// TIA Portal project "Lab4" (V16)

(* hardware
DEVICE "S71500/ET200MP station_1"  S7-1500 station
   slot 0: "PM 190W 120/230VAC"  PM 190W 120/230VAC  6EP1333-4BA00
   slot 0: "Perfil soporte_0"  Rack  6ES7 590-1***0-0AA0
   slot 1: "PLC_1"  CPU 1516-3 PN/DP  6ES7 516-3AN01-0AB0  V1.8
      slot 3: "Display de la CPU_1"  6ES7591-1BA00-0AA0
      slot 32768: "Interfaz PROFINET_1"  X1
         slot 32769: "Puerto_1"  X1 P1
         slot 32770: "Puerto_2"  X1 P2
      slot 33024: "Interfaz PROFINET_2"  X2
         slot 33025: "Puerto_1"  X2 P1
      slot 33280: "Interfaz DP_1"  X3
   slot 2: "DI 32x24VDC HF_1"  DI 32x24VDC HF  6ES7 521-1BL00-0AB0  V1.0
   slot 3: "DQ 32x24VDC/0.5A ST_1"  DQ 32x24VDC/0.5A ST  6ES7 522-1BL00-0AB0  V1.0
   slot 4: "AI 8xU/I/RTD/TC ST_1"  AI 8xU/I/RTD/TC ST  6ES7 531-7KF00-0AB0  V1.0
   slot 5: "AQ 4xU/I ST_1"  AQ 4xU/I ST  6ES7 532-5HD00-0AB0  V1.0
*)

// ===== PLC "PLC_1"  CPU 1516-3 PN/DP =====

VAR_GLOBAL   // PLC tag table "Tabla de variables estándar"
   "10001" AT %M0.0 : Bool;
   "10003" AT %M0.2 : Bool;
   "ON2" AT %M100.0 : Bool;
   "10005" AT %M0.4 : Bool;
   "OFF14-15-ONMP1-CUA" AT %M201.0 : Bool;
   "OFFMP1-CUA" AT %M202.0 : Bool;
   "OFFMP2YONMP1-C1" AT %M212.0 : Bool;
   "ON1YON4" AT %M101.0 : Bool;
   "10004" AT %M0.3 : Bool;
   "OFF1YOFF4" AT %M102.0 : Bool;
   "OFF2" AT %M103.0 : Bool;
   "ON1YON3" AT %M104.0 : Bool;
   "OFF1YON4" AT %M105.0 : Bool;
   "OFF3YOFF4" AT %M106.0 : Bool;
   "2" AT %Q0.1 : Bool;
   "1" AT %Q0.0 : Bool;
   "4" AT %Q0.3 : Bool;
   "3" AT %Q0.2 : Bool;
   "10002" AT %M0.1 : Bool;
   "10006" AT %M0.5 : Bool;
   "10028" AT %I0.0 : Bool;
   "10021" AT %I0.4 : Bool;
   "10023" AT %I0.1 : Bool;
   "10025" AT %I0.5 : Bool;
   "ON9-10-15" AT %M210.0 : Bool;
   "OFF8" AT %M116.0 : Bool;
   "OFFMP1-C1" AT %M213.0 : Bool;
   "10" AT %Q1.0 : Bool;
   "9" AT %Q0.7 : Bool;
   "15" AT %Q1.5 : Bool;
   "10010" AT %M0.7 : Bool;
   "10011" AT %M1.0 : Bool;
   "10012" AT %M1.1 : Bool;
   "10009" AT %M0.6 : Bool;
   "OFF9-10-15YONMP2-C1" AT %M211.0 : Bool;
   "OFF15-13-12-11YONMP2-C2" AT %M216.0 : Bool;
   "ON8YON5" AT %M110.0 : Bool;
   "OFF8YOFF5" AT %M111.0 : Bool;
   "ON6" AT %M112.0 : Bool;
   "ON5" AT %M113.0 : Bool;
   "ON8YOFF5" AT %M114.0 : Bool;
   "OFF6" AT %M115.0 : Bool;
   "5" AT %Q0.4 : Bool;
   "8" AT %Q0.6 : Bool;
   "6" AT %Q0.5 : Bool;
   "10022" AT %I0.3 : Bool;
   "14" AT %Q1.4 : Bool;
   "ON14-15" AT %M200.0 : Bool;
   "10024" AT %I0.2 : Bool;
   "ON15-11-12-13" AT %M215.0 : Bool;
   "OFFMP1-C2" AT %M218.0 : Bool;
   "OFFMP2YONMP1-C2" AT %M217.0 : Bool;
   "11" AT %Q1.1 : Bool;
   "12" AT %Q1.2 : Bool;
   "13" AT %Q1.3 : Bool;
   "RUN" AT %M2.0 : Bool;
   "STOP" AT %M2.1 : Bool;
   "Inic_Proce" AT %M60.0 : Bool;
   "Sec_Cuadrado" AT %M60.1 : Bool;
   "Aux1" AT %M300.0 : Bool;
   "Sec_Cilindro1" AT %M60.2 : Bool;
   "Sec_Cilindro2" AT %M60.3 : Bool;
   "Aux2" AT %M300.1 : Bool;
   "15AUX" AT %M500.0 : Bool;
   "Tag_1" AT %MB3 : Byte;
END_VAR

// folder: System blocks/Program resources

DATA_BLOCK "IEC_Counter_0_DB"   // DB1
{ S7_Optimized_Access := 'TRUE' }
AUTHOR : Simatic
FAMILY : IEC
NAME : CNTR
VERSION : 1.0
// stored: InstanceOfName IEC_COUNTER
"IEC_COUNTER"
BEGIN
END_DATA_BLOCK

// folder: (top level)

FUNCTION "MP1" : Void   // FC1, LAD
{ S7_Optimized_Access := 'TRUE' }
VERSION : 0.1
BEGIN

REGION Network 1
   // MP1
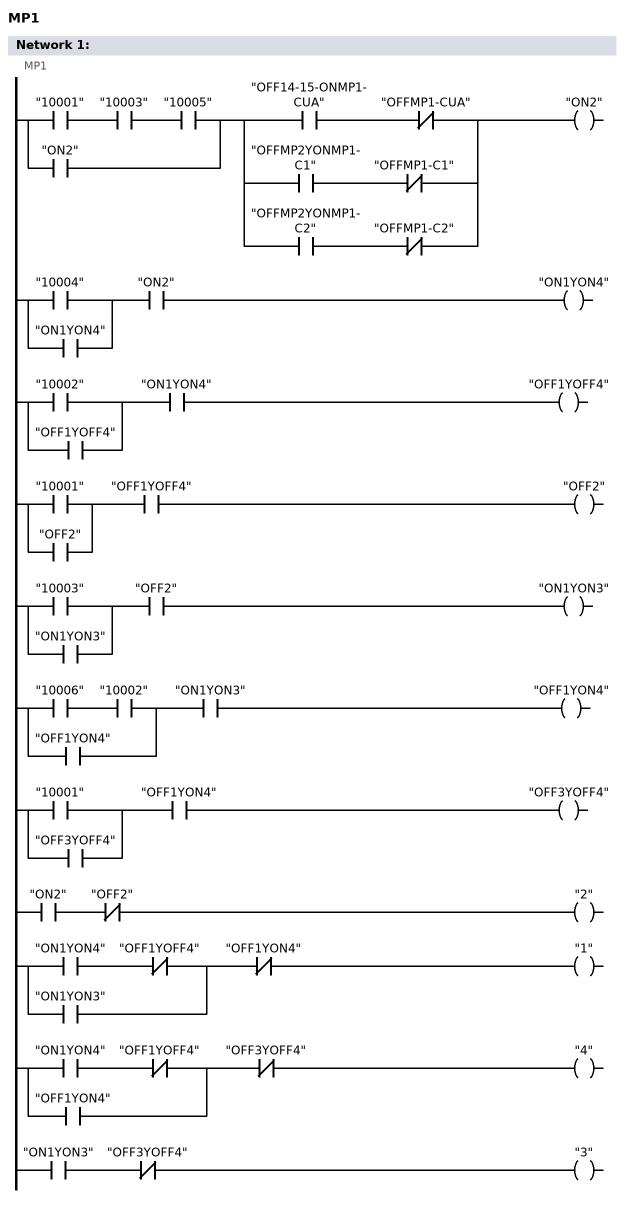
   RUNG wire#powerrail
      Contact( "10001" )
      Contact( "10003" )
      Contact( "10005" )
      wire#w1
      Contact( "OFF14-15-ONMP1-CUA" )
      I_Contact( "OFFMP1-CUA" )
      wire#w2
      Coil( "ON2" )
   END_RUNG
   RUNG wire#powerrail
      Contact( "ON2" )
   END_RUNG wire#w1
   RUNG wire#w1
      Contact( "OFFMP2YONMP1-C1" )
      I_Contact( "OFFMP1-C1" )
   END_RUNG wire#w2
   RUNG wire#w1
      Contact( "OFFMP2YONMP1-C2" )
      I_Contact( "OFFMP1-C2" )
   END_RUNG wire#w2
   RUNG wire#powerrail
      Contact( "10004" )
      wire#w3
      Contact( "ON2" )
      Coil( "ON1YON4" )
   END_RUNG
   RUNG wire#powerrail
      Contact( "ON1YON4" )
   END_RUNG wire#w3
   RUNG wire#powerrail
      Contact( "10002" )
      wire#w4
      Contact( "ON1YON4" )
      Coil( "OFF1YOFF4" )
   END_RUNG
   RUNG wire#powerrail
      Contact( "OFF1YOFF4" )
   END_RUNG wire#w4
   RUNG wire#powerrail
      Contact( "10001" )
      wire#w5
      Contact( "OFF1YOFF4" )
      Coil( "OFF2" )
   END_RUNG
   RUNG wire#powerrail
      Contact( "OFF2" )
   END_RUNG wire#w5
   RUNG wire#powerrail
      Contact( "10003" )
      wire#w6
      Contact( "OFF2" )
      Coil( "ON1YON3" )
   END_RUNG
   RUNG wire#powerrail
      Contact( "ON1YON3" )
   END_RUNG wire#w6
   RUNG wire#powerrail
      Contact( "10006" )
      Contact( "10002" )
      wire#w7
      Contact( "ON1YON3" )
      Coil( "OFF1YON4" )
   END_RUNG
   RUNG wire#powerrail
      Contact( "OFF1YON4" )
   END_RUNG wire#w7
   RUNG wire#powerrail
      Contact( "10001" )
      wire#w8
      Contact( "OFF1YON4" )
      Coil( "OFF3YOFF4" )
   END_RUNG
   RUNG wire#powerrail
      Contact( "OFF3YOFF4" )
   END_RUNG wire#w8
   RUNG wire#powerrail
      Contact( "ON2" )
      I_Contact( "OFF2" )
      Coil( "2" )
   END_RUNG
   RUNG wire#powerrail
      Contact( "ON1YON4" )
      I_Contact( "OFF1YOFF4" )
      wire#w9
      I_Contact( "OFF1YON4" )
      Coil( "1" )
   END_RUNG
   RUNG wire#powerrail
      Contact( "ON1YON3" )
   END_RUNG wire#w9
   RUNG wire#powerrail
      Contact( "ON1YON4" )
      I_Contact( "OFF1YOFF4" )
      wire#w10
      I_Contact( "OFF3YOFF4" )
      Coil( "4" )
   END_RUNG
   RUNG wire#powerrail
      Contact( "OFF1YON4" )
   END_RUNG wire#w10
   RUNG wire#powerrail
      Contact( "ON1YON3" )
      I_Contact( "OFF3YOFF4" )
      Coil( "3" )
   END_RUNG
   // the same network as SCL:
   "ON2" := (("10001" AND "10003" AND "10005") OR "ON2") AND (("OFF14-15-ONMP1-CUA" AND NOT "OFFMP1-CUA") OR ("OFFMP2YONMP1-C1" AND NOT "OFFMP1-C1") OR ("OFFMP2YONMP1-C2" AND NOT "OFFMP1-C2"));
   "ON1YON4" := ("10004" OR "ON1YON4") AND "ON2";
   "OFF1YOFF4" := ("10002" OR "OFF1YOFF4") AND "ON1YON4";
   "OFF2" := ("10001" OR "OFF2") AND "OFF1YOFF4";
   "ON1YON3" := ("10003" OR "ON1YON3") AND "OFF2";
   "OFF1YON4" := (("10006" AND "10002") OR "OFF1YON4") AND "ON1YON3";
   "OFF3YOFF4" := ("10001" OR "OFF3YOFF4") AND "OFF1YON4";
   "2" := "ON2" AND NOT "OFF2";
   "1" := (("ON1YON4" AND NOT "OFF1YOFF4") OR "ON1YON3") AND NOT "OFF1YON4";
   "4" := (("ON1YON4" AND NOT "OFF1YOFF4") OR "OFF1YON4") AND NOT "OFF3YOFF4";
   "3" := "ON1YON3" AND NOT "OFF3YOFF4";
END_REGION
END_FUNCTION

FUNCTION "MP2" : Void   // FC2, LAD
{ S7_Optimized_Access := 'TRUE' }
VERSION : 0.1
BEGIN

REGION Network 1
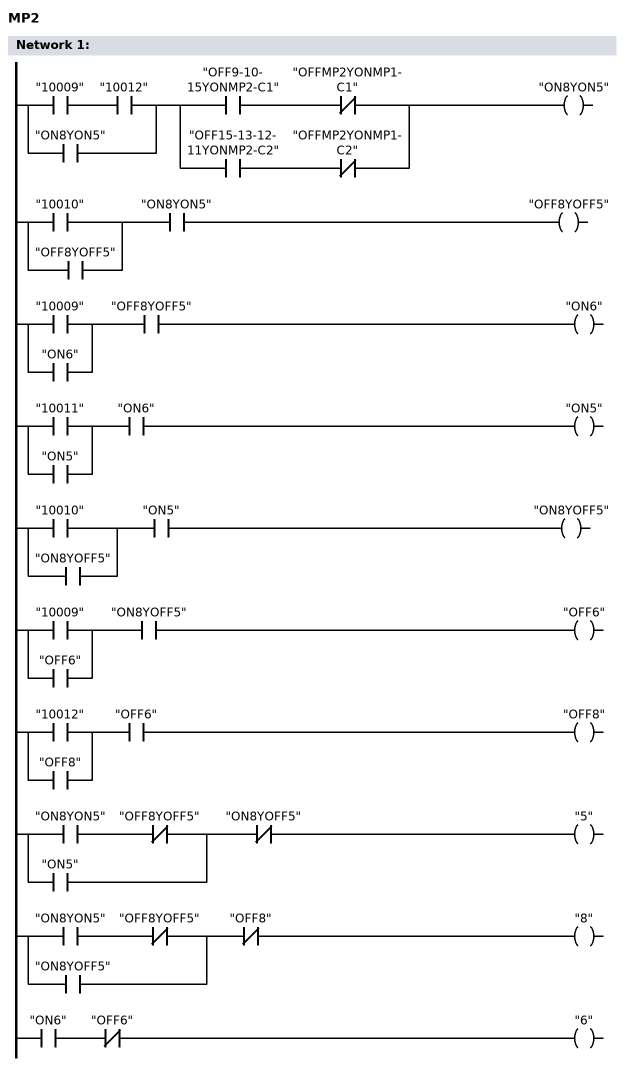
   RUNG wire#powerrail
      Contact( "10009" )
      Contact( "10012" )
      wire#w1
      Contact( "OFF9-10-15YONMP2-C1" )
      I_Contact( "OFFMP2YONMP1-C1" )
      wire#w2
      Coil( "ON8YON5" )
   END_RUNG
   RUNG wire#powerrail
      Contact( "ON8YON5" )
   END_RUNG wire#w1
   RUNG wire#w1
      Contact( "OFF15-13-12-11YONMP2-C2" )
      I_Contact( "OFFMP2YONMP1-C2" )
   END_RUNG wire#w2
   RUNG wire#powerrail
      Contact( "10010" )
      wire#w3
      Contact( "ON8YON5" )
      Coil( "OFF8YOFF5" )
   END_RUNG
   RUNG wire#powerrail
      Contact( "OFF8YOFF5" )
   END_RUNG wire#w3
   RUNG wire#powerrail
      Contact( "10009" )
      wire#w4
      Contact( "OFF8YOFF5" )
      Coil( "ON6" )
   END_RUNG
   RUNG wire#powerrail
      Contact( "ON6" )
   END_RUNG wire#w4
   RUNG wire#powerrail
      Contact( "10011" )
      wire#w5
      Contact( "ON6" )
      Coil( "ON5" )
   END_RUNG
   RUNG wire#powerrail
      Contact( "ON5" )
   END_RUNG wire#w5
   RUNG wire#powerrail
      Contact( "10010" )
      wire#w6
      Contact( "ON5" )
      Coil( "ON8YOFF5" )
   END_RUNG
   RUNG wire#powerrail
      Contact( "ON8YOFF5" )
   END_RUNG wire#w6
   RUNG wire#powerrail
      Contact( "10009" )
      wire#w7
      Contact( "ON8YOFF5" )
      Coil( "OFF6" )
   END_RUNG
   RUNG wire#powerrail
      Contact( "OFF6" )
   END_RUNG wire#w7
   RUNG wire#powerrail
      Contact( "10012" )
      wire#w8
      Contact( "OFF6" )
      Coil( "OFF8" )
   END_RUNG
   RUNG wire#powerrail
      Contact( "OFF8" )
   END_RUNG wire#w8
   RUNG wire#powerrail
      Contact( "ON8YON5" )
      I_Contact( "OFF8YOFF5" )
      wire#w9
      I_Contact( "ON8YOFF5" )
      Coil( "5" )
   END_RUNG
   RUNG wire#powerrail
      Contact( "ON5" )
   END_RUNG wire#w9
   RUNG wire#powerrail
      Contact( "ON8YON5" )
      I_Contact( "OFF8YOFF5" )
      wire#w10
      I_Contact( "OFF8" )
      Coil( "8" )
   END_RUNG
   RUNG wire#powerrail
      Contact( "ON8YOFF5" )
   END_RUNG wire#w10
   RUNG wire#powerrail
      Contact( "ON6" )
      I_Contact( "OFF6" )
      Coil( "6" )
   END_RUNG
   // the same network as SCL:
   "ON8YON5" := (("10009" AND "10012") OR "ON8YON5") AND (("OFF9-10-15YONMP2-C1" AND NOT "OFFMP2YONMP1-C1") OR ("OFF15-13-12-11YONMP2-C2" AND NOT "OFFMP2YONMP1-C2"));
   "OFF8YOFF5" := ("10010" OR "OFF8YOFF5") AND "ON8YON5";
   "ON6" := ("10009" OR "ON6") AND "OFF8YOFF5";
   "ON5" := ("10011" OR "ON5") AND "ON6";
   "ON8YOFF5" := ("10010" OR "ON8YOFF5") AND "ON5";
   "OFF6" := ("10009" OR "OFF6") AND "ON8YOFF5";
   "OFF8" := ("10012" OR "OFF8") AND "OFF6";
   "5" := (("ON8YON5" AND NOT "OFF8YOFF5") OR "ON5") AND NOT "ON8YOFF5";
   "8" := (("ON8YON5" AND NOT "OFF8YOFF5") OR "ON8YOFF5") AND NOT "OFF8";
   "6" := "ON6" AND NOT "OFF6";
END_REGION
END_FUNCTION

FUNCTION "CUADRADOS" : Void   // FC3, LAD
{ S7_Optimized_Access := 'TRUE' }
VERSION : 0.1
BEGIN

REGION Network 1
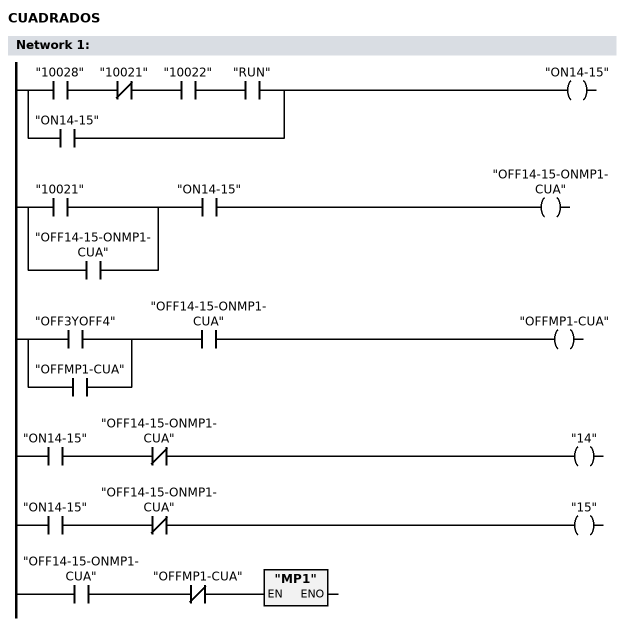
   RUNG wire#powerrail
      Contact( "10028" )
      I_Contact( "10021" )
      Contact( "10022" )
      Contact( "RUN" )
      wire#w1
      Coil( "ON14-15" )
   END_RUNG
   RUNG wire#powerrail
      Contact( "ON14-15" )
   END_RUNG wire#w1
   RUNG wire#powerrail
      Contact( "10021" )
      wire#w2
      Contact( "ON14-15" )
      Coil( "OFF14-15-ONMP1-CUA" )
   END_RUNG
   RUNG wire#powerrail
      Contact( "OFF14-15-ONMP1-CUA" )
   END_RUNG wire#w2
   RUNG wire#powerrail
      Contact( "OFF3YOFF4" )
      wire#w3
      Contact( "OFF14-15-ONMP1-CUA" )
      Coil( "OFFMP1-CUA" )
   END_RUNG
   RUNG wire#powerrail
      Contact( "OFFMP1-CUA" )
   END_RUNG wire#w3
   RUNG wire#powerrail
      Contact( "ON14-15" )
      I_Contact( "OFF14-15-ONMP1-CUA" )
      Coil( "14" )
   END_RUNG
   RUNG wire#powerrail
      Contact( "ON14-15" )
      I_Contact( "OFF14-15-ONMP1-CUA" )
      Coil( "15" )
   END_RUNG
   RUNG wire#powerrail
      Contact( "OFF14-15-ONMP1-CUA" )
      I_Contact( "OFFMP1-CUA" )
      "MP1"()
   END_RUNG
   // the same network as SCL:
   "ON14-15" := ("10028" AND NOT "10021" AND "10022" AND "RUN") OR "ON14-15";
   "OFF14-15-ONMP1-CUA" := ("10021" OR "OFF14-15-ONMP1-CUA") AND "ON14-15";
   "OFFMP1-CUA" := ("OFF3YOFF4" OR "OFFMP1-CUA") AND "OFF14-15-ONMP1-CUA";
   "14" := "ON14-15" AND NOT "OFF14-15-ONMP1-CUA";
   "15" := "ON14-15" AND NOT "OFF14-15-ONMP1-CUA";
   IF "OFF14-15-ONMP1-CUA" AND NOT "OFFMP1-CUA" THEN "MP1"(); END_IF;
END_REGION
END_FUNCTION

FUNCTION "CILINDRO1" : Void   // FC4, LAD
{ S7_Optimized_Access := 'TRUE' }
VERSION : 0.1
BEGIN

REGION Network 1
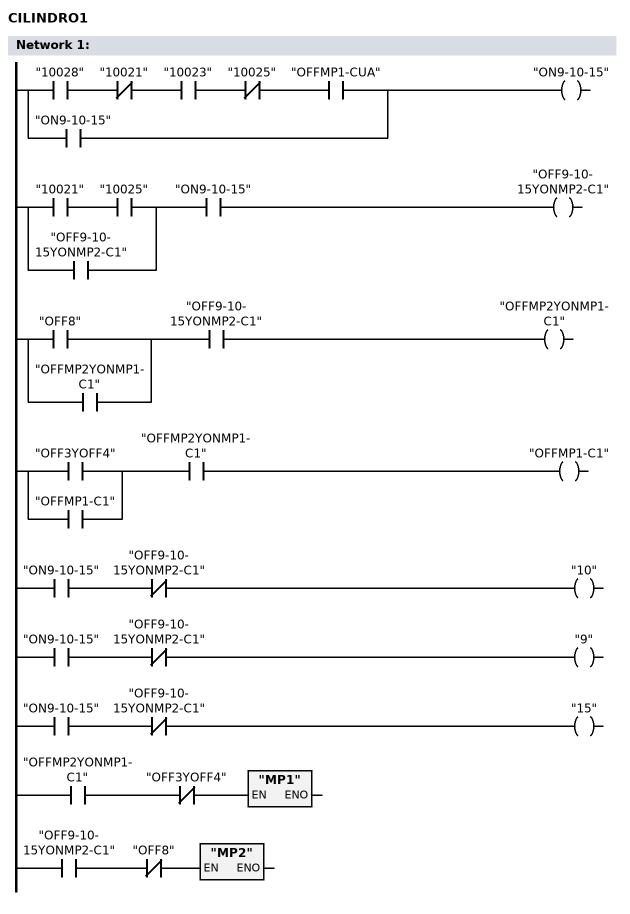
   RUNG wire#powerrail
      Contact( "10028" )
      I_Contact( "10021" )
      Contact( "10023" )
      I_Contact( "10025" )
      Contact( "OFFMP1-CUA" )
      wire#w1
      Coil( "ON9-10-15" )
   END_RUNG
   RUNG wire#powerrail
      Contact( "ON9-10-15" )
   END_RUNG wire#w1
   RUNG wire#powerrail
      Contact( "10021" )
      Contact( "10025" )
      wire#w2
      Contact( "ON9-10-15" )
      Coil( "OFF9-10-15YONMP2-C1" )
   END_RUNG
   RUNG wire#powerrail
      Contact( "OFF9-10-15YONMP2-C1" )
   END_RUNG wire#w2
   RUNG wire#powerrail
      Contact( "OFF8" )
      wire#w3
      Contact( "OFF9-10-15YONMP2-C1" )
      Coil( "OFFMP2YONMP1-C1" )
   END_RUNG
   RUNG wire#powerrail
      Contact( "OFFMP2YONMP1-C1" )
   END_RUNG wire#w3
   RUNG wire#powerrail
      Contact( "OFF3YOFF4" )
      wire#w4
      Contact( "OFFMP2YONMP1-C1" )
      Coil( "OFFMP1-C1" )
   END_RUNG
   RUNG wire#powerrail
      Contact( "OFFMP1-C1" )
   END_RUNG wire#w4
   RUNG wire#powerrail
      Contact( "ON9-10-15" )
      I_Contact( "OFF9-10-15YONMP2-C1" )
      Coil( "10" )
   END_RUNG
   RUNG wire#powerrail
      Contact( "ON9-10-15" )
      I_Contact( "OFF9-10-15YONMP2-C1" )
      Coil( "9" )
   END_RUNG
   RUNG wire#powerrail
      Contact( "ON9-10-15" )
      I_Contact( "OFF9-10-15YONMP2-C1" )
      Coil( "15" )
   END_RUNG
   RUNG wire#powerrail
      Contact( "OFFMP2YONMP1-C1" )
      I_Contact( "OFF3YOFF4" )
      "MP1"()
   END_RUNG
   RUNG wire#powerrail
      Contact( "OFF9-10-15YONMP2-C1" )
      I_Contact( "OFF8" )
      "MP2"()
   END_RUNG
   // the same network as SCL:
   "ON9-10-15" := ("10028" AND NOT "10021" AND "10023" AND NOT "10025" AND "OFFMP1-CUA") OR "ON9-10-15";
   "OFF9-10-15YONMP2-C1" := (("10021" AND "10025") OR "OFF9-10-15YONMP2-C1") AND "ON9-10-15";
   "OFFMP2YONMP1-C1" := ("OFF8" OR "OFFMP2YONMP1-C1") AND "OFF9-10-15YONMP2-C1";
   "OFFMP1-C1" := ("OFF3YOFF4" OR "OFFMP1-C1") AND "OFFMP2YONMP1-C1";
   "10" := "ON9-10-15" AND NOT "OFF9-10-15YONMP2-C1";
   "9" := "ON9-10-15" AND NOT "OFF9-10-15YONMP2-C1";
   "15" := "ON9-10-15" AND NOT "OFF9-10-15YONMP2-C1";
   IF "OFFMP2YONMP1-C1" AND NOT "OFF3YOFF4" THEN "MP1"(); END_IF;
   IF "OFF9-10-15YONMP2-C1" AND NOT "OFF8" THEN "MP2"(); END_IF;
END_REGION
END_FUNCTION

FUNCTION "CILINDRO2" : Void   // FC5, LAD
{ S7_Optimized_Access := 'TRUE' }
VERSION : 0.1
BEGIN

REGION Network 1
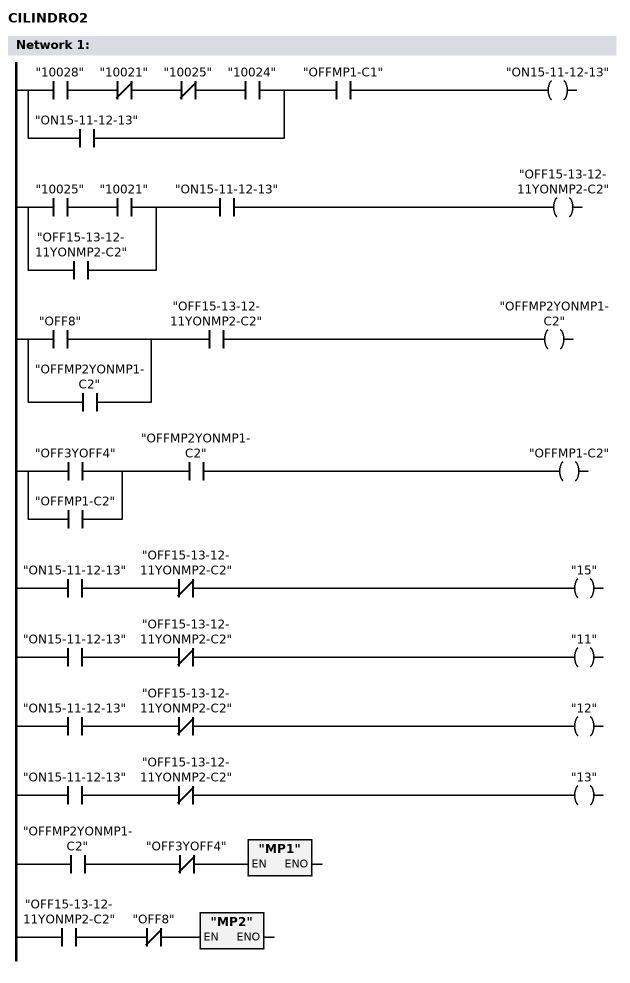
   RUNG wire#powerrail
      Contact( "10028" )
      I_Contact( "10021" )
      I_Contact( "10025" )
      Contact( "10024" )
      wire#w1
      Contact( "OFFMP1-C1" )
      Coil( "ON15-11-12-13" )
   END_RUNG
   RUNG wire#powerrail
      Contact( "ON15-11-12-13" )
   END_RUNG wire#w1
   RUNG wire#powerrail
      Contact( "10025" )
      Contact( "10021" )
      wire#w2
      Contact( "ON15-11-12-13" )
      Coil( "OFF15-13-12-11YONMP2-C2" )
   END_RUNG
   RUNG wire#powerrail
      Contact( "OFF15-13-12-11YONMP2-C2" )
   END_RUNG wire#w2
   RUNG wire#powerrail
      Contact( "OFF8" )
      wire#w3
      Contact( "OFF15-13-12-11YONMP2-C2" )
      Coil( "OFFMP2YONMP1-C2" )
   END_RUNG
   RUNG wire#powerrail
      Contact( "OFFMP2YONMP1-C2" )
   END_RUNG wire#w3
   RUNG wire#powerrail
      Contact( "OFF3YOFF4" )
      wire#w4
      Contact( "OFFMP2YONMP1-C2" )
      Coil( "OFFMP1-C2" )
   END_RUNG
   RUNG wire#powerrail
      Contact( "OFFMP1-C2" )
   END_RUNG wire#w4
   RUNG wire#powerrail
      Contact( "ON15-11-12-13" )
      I_Contact( "OFF15-13-12-11YONMP2-C2" )
      Coil( "15" )
   END_RUNG
   RUNG wire#powerrail
      Contact( "ON15-11-12-13" )
      I_Contact( "OFF15-13-12-11YONMP2-C2" )
      Coil( "11" )
   END_RUNG
   RUNG wire#powerrail
      Contact( "ON15-11-12-13" )
      I_Contact( "OFF15-13-12-11YONMP2-C2" )
      Coil( "12" )
   END_RUNG
   RUNG wire#powerrail
      Contact( "ON15-11-12-13" )
      I_Contact( "OFF15-13-12-11YONMP2-C2" )
      Coil( "13" )
   END_RUNG
   RUNG wire#powerrail
      Contact( "OFFMP2YONMP1-C2" )
      I_Contact( "OFF3YOFF4" )
      "MP1"()
   END_RUNG
   RUNG wire#powerrail
      Contact( "OFF15-13-12-11YONMP2-C2" )
      I_Contact( "OFF8" )
      "MP2"()
   END_RUNG
   // the same network as SCL:
   "ON15-11-12-13" := (("10028" AND NOT "10021" AND NOT "10025" AND "10024") OR "ON15-11-12-13") AND "OFFMP1-C1";
   "OFF15-13-12-11YONMP2-C2" := (("10025" AND "10021") OR "OFF15-13-12-11YONMP2-C2") AND "ON15-11-12-13";
   "OFFMP2YONMP1-C2" := ("OFF8" OR "OFFMP2YONMP1-C2") AND "OFF15-13-12-11YONMP2-C2";
   "OFFMP1-C2" := ("OFF3YOFF4" OR "OFFMP1-C2") AND "OFFMP2YONMP1-C2";
   "15" := "ON15-11-12-13" AND NOT "OFF15-13-12-11YONMP2-C2";
   "11" := "ON15-11-12-13" AND NOT "OFF15-13-12-11YONMP2-C2";
   "12" := "ON15-11-12-13" AND NOT "OFF15-13-12-11YONMP2-C2";
   "13" := "ON15-11-12-13" AND NOT "OFF15-13-12-11YONMP2-C2";
   IF "OFFMP2YONMP1-C2" AND NOT "OFF3YOFF4" THEN "MP1"(); END_IF;
   IF "OFF15-13-12-11YONMP2-C2" AND NOT "OFF8" THEN "MP2"(); END_IF;
END_REGION
END_FUNCTION

FUNCTION "SECUENCIA" : Void   // FC6, LAD
{ S7_Optimized_Access := 'TRUE' }
VERSION : 0.1
   VAR_TEMP
      numero : Int;
      Num : Int;
   END_VAR
   VAR_TEMP   // added for the SCL form of the ladder/FBD networks
      _w1 : Bool;
   END_VAR
BEGIN

REGION Network 1
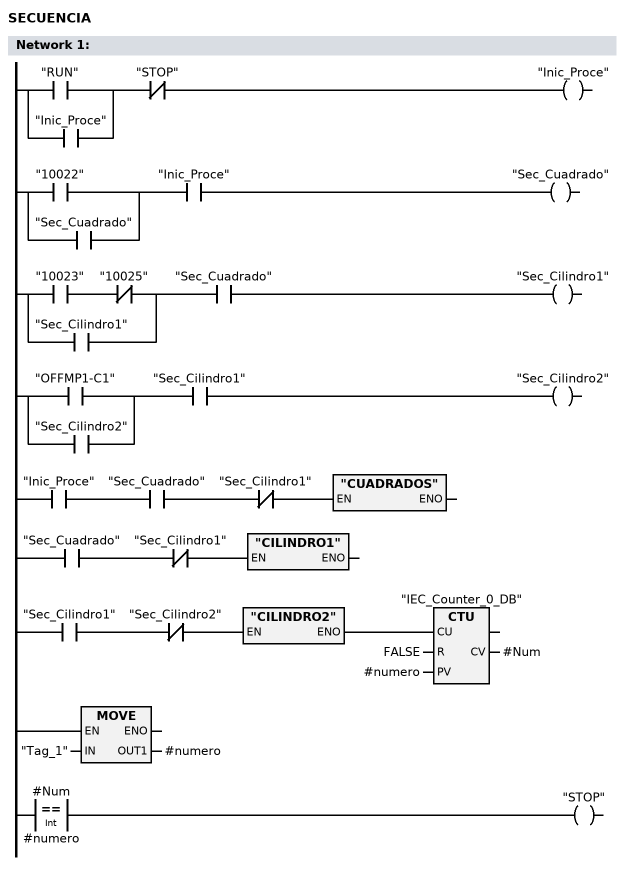
   "Inic_Proce" := ("RUN" OR "Inic_Proce") AND NOT "STOP";
   "Sec_Cuadrado" := ("10022" OR "Sec_Cuadrado") AND "Inic_Proce";
   "Sec_Cilindro1" := (("10023" AND NOT "10025") OR "Sec_Cilindro1") AND "Sec_Cuadrado";
   "Sec_Cilindro2" := ("OFFMP1-C1" OR "Sec_Cilindro2") AND "Sec_Cilindro1";
   IF "Inic_Proce" AND "Sec_Cuadrado" AND NOT "Sec_Cilindro1" THEN "CUADRADOS"(); END_IF;
   IF "Sec_Cuadrado" AND NOT "Sec_Cilindro1" THEN "CILINDRO1"(); END_IF;
   "CILINDRO2"(EN := "Sec_Cilindro1" AND NOT "Sec_Cilindro2", ENO => #_w1);
   "IEC_Counter_0_DB".CTU(CU := #_w1, R := FALSE, PV := #numero, CV => #Num);
   #numero := "Tag_1";
   "STOP" := #Num = #numero;
END_REGION
END_FUNCTION

ORGANIZATION_BLOCK "Main"   // OB1, LAD, ProgramCycle
TITLE = "Main Program Sweep (Cycle)"
{ S7_Optimized_Access := 'TRUE' }
VERSION : 0.1
   VAR_INPUT
      Initial_Call : Bool;   // Initial call of this OB
      Remanence : Bool;   // =True, if remanent data are available
   END_VAR
   VAR_TEMP   // added for the SCL form of the ladder/FBD networks
      _w1 : Bool;
      _w2 : Bool;
      _w3 : Bool;
      _w4 : Bool;
      _w5 : Bool;
   END_VAR
BEGIN

REGION Network 1
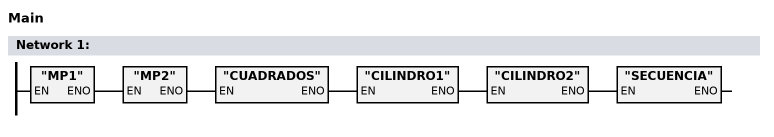
   RUNG wire#powerrail
      "MP1"()
      "MP2"()
      "CUADRADOS"()
      "CILINDRO1"()
      "CILINDRO2"()
      "SECUENCIA"()
   END_RUNG
   // the same network as SCL:
   "MP1"(ENO => #_w1);
   "MP2"(EN := #_w1, ENO => #_w2);
   "CUADRADOS"(EN := #_w2, ENO => #_w3);
   "CILINDRO1"(EN := #_w3, ENO => #_w4);
   "CILINDRO2"(EN := #_w4, ENO => #_w5);
   IF #_w5 THEN "SECUENCIA"(); END_IF;
END_REGION
END_ORGANIZATION_BLOCK